FUNCTION "Conditions_Demarrage" : Bool
{ S7_Optimized_Access := 'TRUE' }
VERSION : 0.1
   VAR_IN_OUT
      Broyeur : "S_Broyage";
   END_VAR


BEGIN
	#Conditions_Demarrage := TRUE;
END_FUNCTION

